// TIA Portal V21 export
FUNCTION "Main paratie" : Void   // FC5001, LAD
{ S7_Optimized_Access := 'TRUE' }
// stored: AutoNumber false, SetENOAutomatically false
   VAR_TEMP
      UscitaPos : Bool;
      UscitaNeg : Bool;
      UscitaVeloce : Bool;
   END_VAR
   VAR CONSTANT
      Disabilitato : Bool := 0;
   END_VAR
BEGIN

REGION Network 1 (SCL): Gestione paratia 1 - Scorta
   "GestParatia"(Abilitazione := True,
                 SetpointAuto := 50.0,
                 ForzaTuttoPos := #Disabilitato,
                 ForzaTuttoNeg := #Disabilitato,
                 FinecorsaPos := False,
                 FinecorsaNeg := False,
                 BypassFinecorsa := #Disabilitato,
                 K_Zona := "K_Zona_Esempio",
                 K_Paratia := "K_Paratia_Esempio",
                 K_Analogica := "K_Analogica_Esempio",
                 UscitaPos := #UscitaPos,
                 UscitaNeg := #UscitaNeg,
                 UsctaVeloce := #UscitaVeloce);
END_REGION
END_FUNCTION
